Fanuc KAREL source: KT00802.KL

PROGRAM KT00802
%NOLOCKGROUP
VAR
  H1: ARRAY[2] OF SHORT
  H2: ARRAY[2] OF SHORT
  OUT: INTEGER
BEGIN
  H1[1] = 2
  H2[1] = 3
  H1[1] = 2
  H2[1] = 3
  OUT = EXP(H1[1])
END KT00802
